// TIA Portal V19 export
FUNCTION "INPUT" : Void   // FC1, LAD
{ S7_Optimized_Access := 'TRUE' }
// stored: SetENOAutomatically false
BEGIN

REGION Network 1: "EMG STOP"
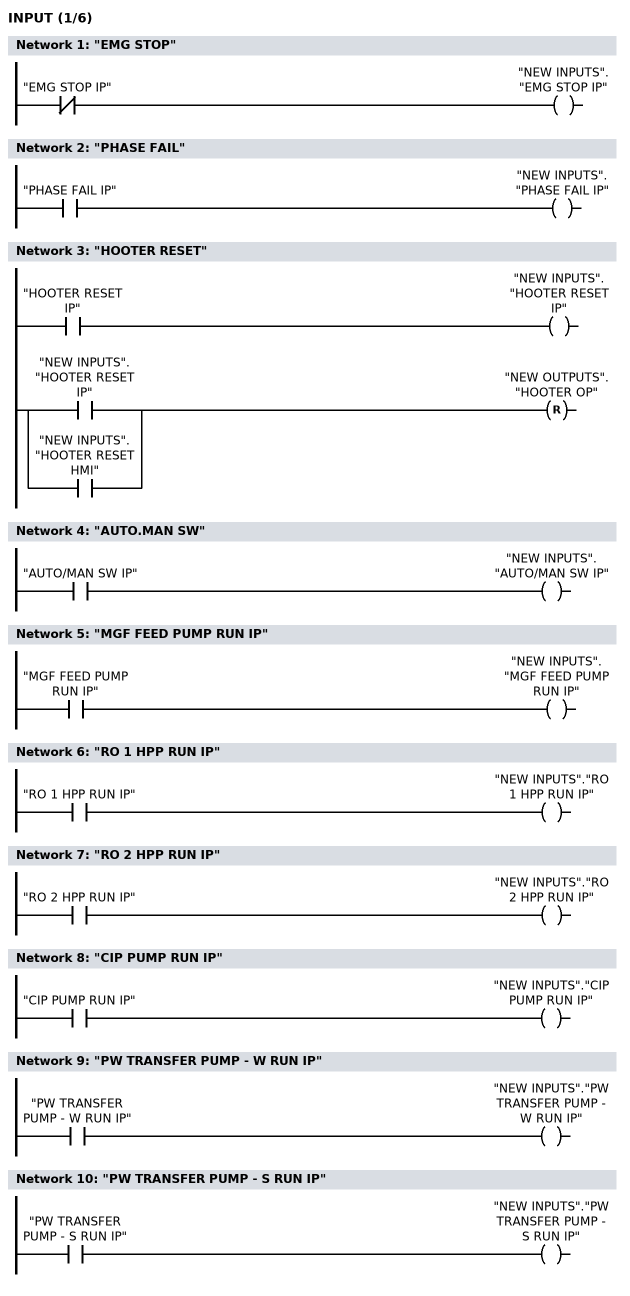
   RUNG wire#powerrail
      I_Contact( "EMG STOP IP" )
      Coil( "NEW INPUTS"."EMG STOP IP" )
   END_RUNG
   // the same network as SCL:
   "NEW INPUTS"."EMG STOP IP" := NOT "EMG STOP IP";
END_REGION

REGION Network 2: "PHASE FAIL"
   RUNG wire#powerrail
      Contact( "PHASE FAIL IP" )
      Coil( "NEW INPUTS"."PHASE FAIL IP" )
   END_RUNG
   // the same network as SCL:
   "NEW INPUTS"."PHASE FAIL IP" := "PHASE FAIL IP";
END_REGION

REGION Network 3: "HOOTER RESET"
   RUNG wire#powerrail
      Contact( "HOOTER RESET IP" )
      Coil( "NEW INPUTS"."HOOTER RESET IP" )
   END_RUNG
   RUNG wire#powerrail
      Contact( "NEW INPUTS"."HOOTER RESET IP" )
      wire#w1
      R_Coil( "NEW OUTPUTS"."HOOTER OP" )
   END_RUNG
   RUNG wire#powerrail
      Contact( "NEW INPUTS"."HOOTER RESET HMI" )
   END_RUNG wire#w1
   // the same network as SCL:
   "NEW INPUTS"."HOOTER RESET IP" := "HOOTER RESET IP";
   IF "NEW INPUTS"."HOOTER RESET IP" OR "NEW INPUTS"."HOOTER RESET HMI" THEN
       "NEW OUTPUTS"."HOOTER OP" := FALSE;
   END_IF;
END_REGION

REGION Network 4: "AUTO.MAN SW"
   RUNG wire#powerrail
      Contact( "AUTO/MAN SW IP" )
      Coil( "NEW INPUTS"."AUTO/MAN SW IP" )
   END_RUNG
   // the same network as SCL:
   "NEW INPUTS"."AUTO/MAN SW IP" := "AUTO/MAN SW IP";
END_REGION

REGION Network 5: "MGF FEED PUMP RUN IP"
   RUNG wire#powerrail
      Contact( "MGF FEED PUMP RUN IP" )
      Coil( "NEW INPUTS"."MGF FEED PUMP RUN IP" )
   END_RUNG
   // the same network as SCL:
   "NEW INPUTS"."MGF FEED PUMP RUN IP" := "MGF FEED PUMP RUN IP";
END_REGION

REGION Network 6: "RO 1 HPP RUN IP"
   RUNG wire#powerrail
      Contact( "RO 1 HPP RUN IP" )
      Coil( "NEW INPUTS"."RO 1 HPP RUN IP" )
   END_RUNG
   // the same network as SCL:
   "NEW INPUTS"."RO 1 HPP RUN IP" := "RO 1 HPP RUN IP";
END_REGION

REGION Network 7: "RO 2 HPP RUN IP"
   RUNG wire#powerrail
      Contact( "RO 2 HPP RUN IP" )
      Coil( "NEW INPUTS"."RO 2 HPP RUN IP" )
   END_RUNG
   // the same network as SCL:
   "NEW INPUTS"."RO 2 HPP RUN IP" := "RO 2 HPP RUN IP";
END_REGION

REGION Network 8: "CIP PUMP RUN IP"
   RUNG wire#powerrail
      Contact( "CIP PUMP RUN IP" )
      Coil( "NEW INPUTS"."CIP PUMP RUN IP" )
   END_RUNG
   // the same network as SCL:
   "NEW INPUTS"."CIP PUMP RUN IP" := "CIP PUMP RUN IP";
END_REGION

REGION Network 9: "PW TRANSFER PUMP - W RUN IP"
   RUNG wire#powerrail
      Contact( "PW TRANSFER PUMP - W RUN IP" )
      Coil( "NEW INPUTS"."PW TRANSFER PUMP - W RUN IP" )
   END_RUNG
   // the same network as SCL:
   "NEW INPUTS"."PW TRANSFER PUMP - W RUN IP" := "PW TRANSFER PUMP - W RUN IP";
END_REGION

REGION Network 10: "PW TRANSFER PUMP - S RUN IP"
   RUNG wire#powerrail
      Contact( "PW TRANSFER PUMP - S RUN IP" )
      Coil( "NEW INPUTS"."PW TRANSFER PUMP - S RUN IP" )
   END_RUNG
   // the same network as SCL:
   "NEW INPUTS"."PW TRANSFER PUMP - S RUN IP" := "PW TRANSFER PUMP - S RUN IP";
END_REGION

REGION Network 11: PW TRANSFER W/P
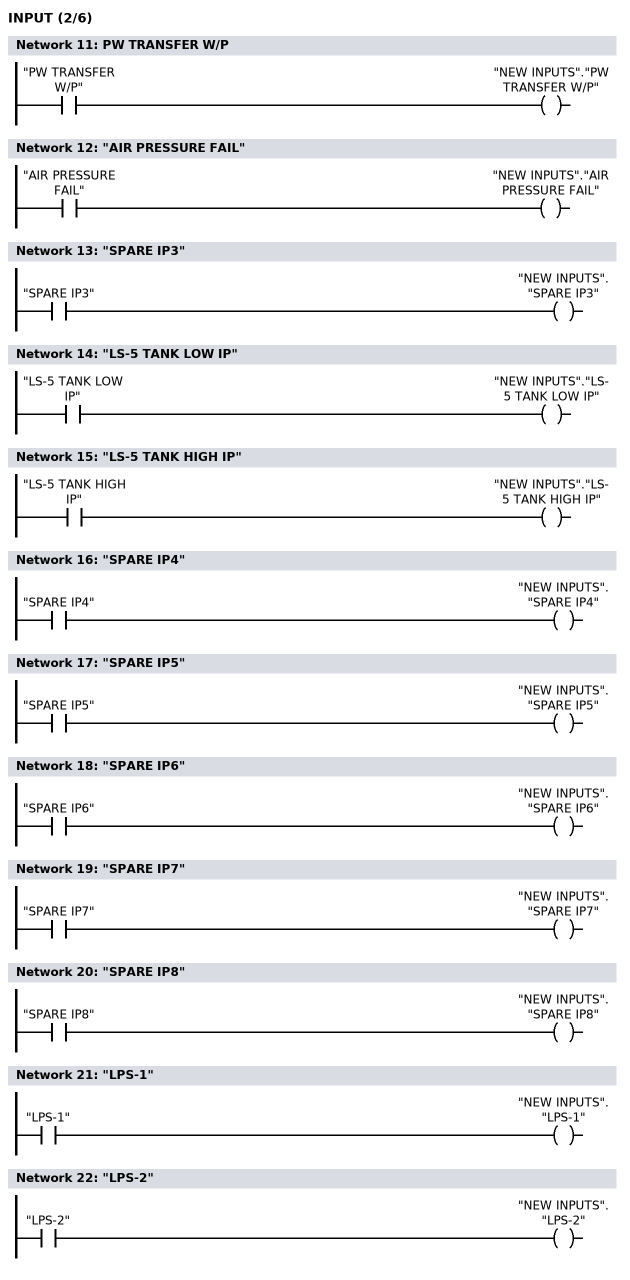
   RUNG wire#powerrail
      Contact( "PW TRANSFER W/P" )
      Coil( "NEW INPUTS"."PW TRANSFER W/P" )
   END_RUNG
   // the same network as SCL:
   "NEW INPUTS"."PW TRANSFER W/P" := "PW TRANSFER W/P";
END_REGION

REGION Network 12: "AIR PRESSURE FAIL"
   RUNG wire#powerrail
      Contact( "AIR PRESSURE FAIL" )
      Coil( "NEW INPUTS"."AIR PRESSURE FAIL" )
   END_RUNG
   // the same network as SCL:
   "NEW INPUTS"."AIR PRESSURE FAIL" := "AIR PRESSURE FAIL";
END_REGION

REGION Network 13: "SPARE IP3"
   RUNG wire#powerrail
      Contact( "SPARE IP3" )
      Coil( "NEW INPUTS"."SPARE IP3" )
   END_RUNG
   // the same network as SCL:
   "NEW INPUTS"."SPARE IP3" := "SPARE IP3";
END_REGION

REGION Network 14: "LS-5 TANK LOW IP"
   RUNG wire#powerrail
      Contact( "LS-5 TANK LOW IP" )
      Coil( "NEW INPUTS"."LS-5 TANK LOW IP" )
   END_RUNG
   // the same network as SCL:
   "NEW INPUTS"."LS-5 TANK LOW IP" := "LS-5 TANK LOW IP";
END_REGION

REGION Network 15: "LS-5 TANK HIGH IP"
   RUNG wire#powerrail
      Contact( "LS-5 TANK HIGH IP" )
      Coil( "NEW INPUTS"."LS-5 TANK HIGH IP" )
   END_RUNG
   // the same network as SCL:
   "NEW INPUTS"."LS-5 TANK HIGH IP" := "LS-5 TANK HIGH IP";
END_REGION

REGION Network 16: "SPARE IP4"
   RUNG wire#powerrail
      Contact( "SPARE IP4" )
      Coil( "NEW INPUTS"."SPARE IP4" )
   END_RUNG
   // the same network as SCL:
   "NEW INPUTS"."SPARE IP4" := "SPARE IP4";
END_REGION

REGION Network 17: "SPARE IP5"
   RUNG wire#powerrail
      Contact( "SPARE IP5" )
      Coil( "NEW INPUTS"."SPARE IP5" )
   END_RUNG
   // the same network as SCL:
   "NEW INPUTS"."SPARE IP5" := "SPARE IP5";
END_REGION

REGION Network 18: "SPARE IP6"
   RUNG wire#powerrail
      Contact( "SPARE IP6" )
      Coil( "NEW INPUTS"."SPARE IP6" )
   END_RUNG
   // the same network as SCL:
   "NEW INPUTS"."SPARE IP6" := "SPARE IP6";
END_REGION

REGION Network 19: "SPARE IP7"
   RUNG wire#powerrail
      Contact( "SPARE IP7" )
      Coil( "NEW INPUTS"."SPARE IP7" )
   END_RUNG
   // the same network as SCL:
   "NEW INPUTS"."SPARE IP7" := "SPARE IP7";
END_REGION

REGION Network 20: "SPARE IP8"
   RUNG wire#powerrail
      Contact( "SPARE IP8" )
      Coil( "NEW INPUTS"."SPARE IP8" )
   END_RUNG
   // the same network as SCL:
   "NEW INPUTS"."SPARE IP8" := "SPARE IP8";
END_REGION

REGION Network 21: "LPS-1"
   RUNG wire#powerrail
      Contact( "LPS-1" )
      Coil( "NEW INPUTS"."LPS-1" )
   END_RUNG
   // the same network as SCL:
   "NEW INPUTS"."LPS-1" := "LPS-1";
END_REGION

REGION Network 22: "LPS-2"
   RUNG wire#powerrail
      Contact( "LPS-2" )
      Coil( "NEW INPUTS"."LPS-2" )
   END_RUNG
   // the same network as SCL:
   "NEW INPUTS"."LPS-2" := "LPS-2";
END_REGION

REGION Network 23: "MGF V-1 OPEN FB"
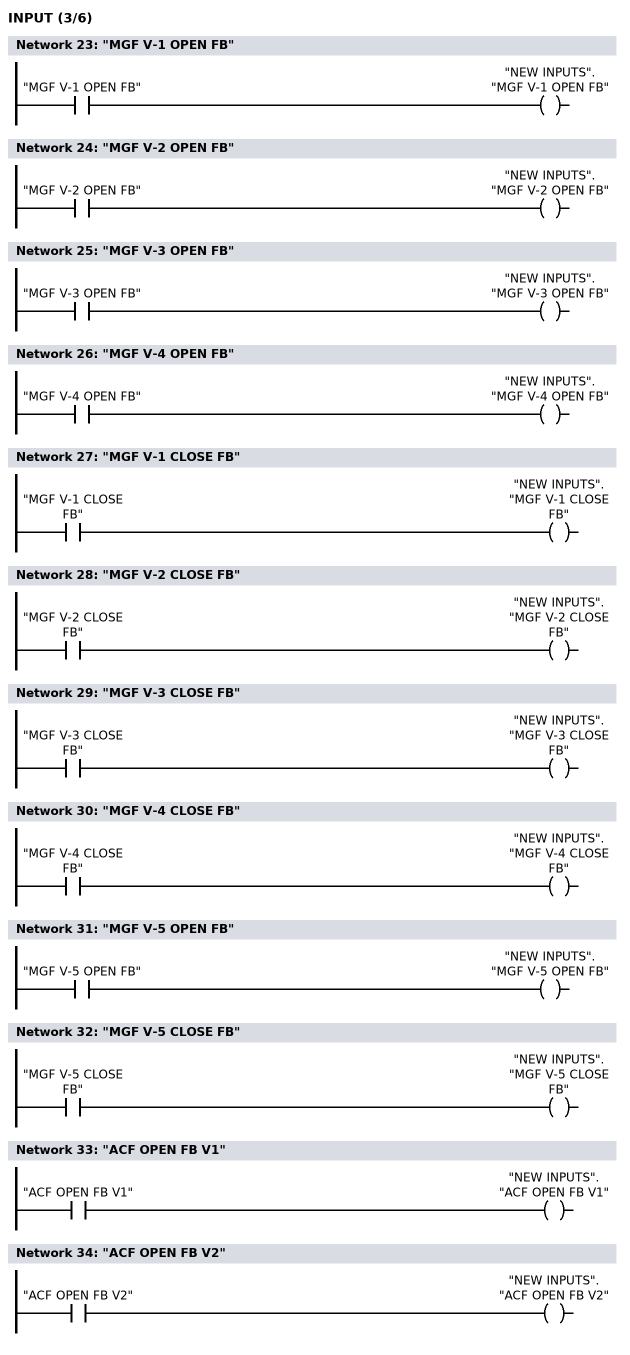
   RUNG wire#powerrail
      Contact( "MGF V-1 OPEN FB" )
      Coil( "NEW INPUTS"."MGF V-1 OPEN FB" )
   END_RUNG
   // the same network as SCL:
   "NEW INPUTS"."MGF V-1 OPEN FB" := "MGF V-1 OPEN FB";
END_REGION

REGION Network 24: "MGF V-2 OPEN FB"
   RUNG wire#powerrail
      Contact( "MGF V-2 OPEN FB" )
      Coil( "NEW INPUTS"."MGF V-2 OPEN FB" )
   END_RUNG
   // the same network as SCL:
   "NEW INPUTS"."MGF V-2 OPEN FB" := "MGF V-2 OPEN FB";
END_REGION

REGION Network 25: "MGF V-3 OPEN FB"
   RUNG wire#powerrail
      Contact( "MGF V-3 OPEN FB" )
      Coil( "NEW INPUTS"."MGF V-3 OPEN FB" )
   END_RUNG
   // the same network as SCL:
   "NEW INPUTS"."MGF V-3 OPEN FB" := "MGF V-3 OPEN FB";
END_REGION

REGION Network 26: "MGF V-4 OPEN FB"
   RUNG wire#powerrail
      Contact( "MGF V-4 OPEN FB" )
      Coil( "NEW INPUTS"."MGF V-4 OPEN FB" )
   END_RUNG
   // the same network as SCL:
   "NEW INPUTS"."MGF V-4 OPEN FB" := "MGF V-4 OPEN FB";
END_REGION

REGION Network 27: "MGF V-1 CLOSE FB"
   RUNG wire#powerrail
      Contact( "MGF V-1 CLOSE FB" )
      Coil( "NEW INPUTS"."MGF V-1 CLOSE FB" )
   END_RUNG
   // the same network as SCL:
   "NEW INPUTS"."MGF V-1 CLOSE FB" := "MGF V-1 CLOSE FB";
END_REGION

REGION Network 28: "MGF V-2 CLOSE FB"
   RUNG wire#powerrail
      Contact( "MGF V-2 CLOSE FB" )
      Coil( "NEW INPUTS"."MGF V-2 CLOSE FB" )
   END_RUNG
   // the same network as SCL:
   "NEW INPUTS"."MGF V-2 CLOSE FB" := "MGF V-2 CLOSE FB";
END_REGION

REGION Network 29: "MGF V-3 CLOSE FB"
   RUNG wire#powerrail
      Contact( "MGF V-3 CLOSE FB" )
      Coil( "NEW INPUTS"."MGF V-3 CLOSE FB" )
   END_RUNG
   // the same network as SCL:
   "NEW INPUTS"."MGF V-3 CLOSE FB" := "MGF V-3 CLOSE FB";
END_REGION

REGION Network 30: "MGF V-4 CLOSE FB"
   RUNG wire#powerrail
      Contact( "MGF V-4 CLOSE FB" )
      Coil( "NEW INPUTS"."MGF V-4 CLOSE FB" )
   END_RUNG
   // the same network as SCL:
   "NEW INPUTS"."MGF V-4 CLOSE FB" := "MGF V-4 CLOSE FB";
END_REGION

REGION Network 31: "MGF V-5 OPEN FB"
   RUNG wire#powerrail
      Contact( "MGF V-5 OPEN FB" )
      Coil( "NEW INPUTS"."MGF V-5 OPEN FB" )
   END_RUNG
   // the same network as SCL:
   "NEW INPUTS"."MGF V-5 OPEN FB" := "MGF V-5 OPEN FB";
END_REGION

REGION Network 32: "MGF V-5 CLOSE FB"
   RUNG wire#powerrail
      Contact( "MGF V-5 CLOSE FB" )
      Coil( "NEW INPUTS"."MGF V-5 CLOSE FB" )
   END_RUNG
   // the same network as SCL:
   "NEW INPUTS"."MGF V-5 CLOSE FB" := "MGF V-5 CLOSE FB";
END_REGION

REGION Network 33: "ACF OPEN FB V1"
   RUNG wire#powerrail
      Contact( "ACF OPEN FB V1" )
      Coil( "NEW INPUTS"."ACF OPEN FB V1" )
   END_RUNG
   // the same network as SCL:
   "NEW INPUTS"."ACF OPEN FB V1" := "ACF OPEN FB V1";
END_REGION

REGION Network 34: "ACF OPEN FB V2"
   RUNG wire#powerrail
      Contact( "ACF OPEN FB V2" )
      Coil( "NEW INPUTS"."ACF OPEN FB V2" )
   END_RUNG
   // the same network as SCL:
   "NEW INPUTS"."ACF OPEN FB V2" := "ACF OPEN FB V2";
END_REGION

REGION Network 35: "ACF OPEN FB V3"
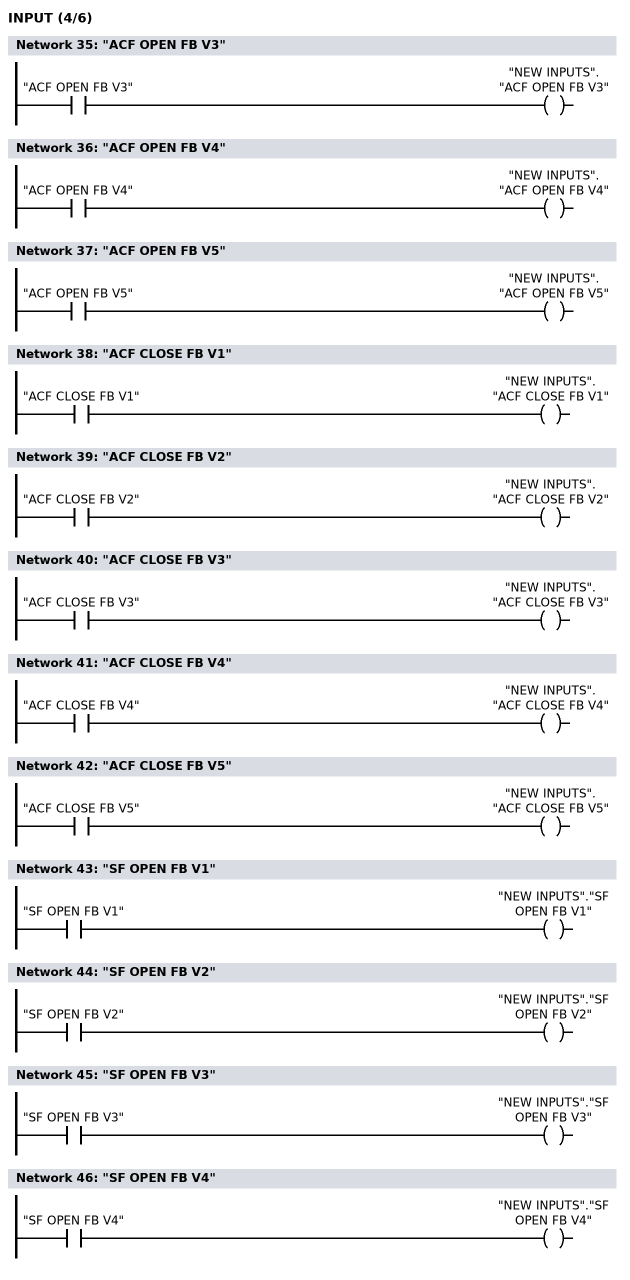
   RUNG wire#powerrail
      Contact( "ACF OPEN FB V3" )
      Coil( "NEW INPUTS"."ACF OPEN FB V3" )
   END_RUNG
   // the same network as SCL:
   "NEW INPUTS"."ACF OPEN FB V3" := "ACF OPEN FB V3";
END_REGION

REGION Network 36: "ACF OPEN FB V4"
   RUNG wire#powerrail
      Contact( "ACF OPEN FB V4" )
      Coil( "NEW INPUTS"."ACF OPEN FB V4" )
   END_RUNG
   // the same network as SCL:
   "NEW INPUTS"."ACF OPEN FB V4" := "ACF OPEN FB V4";
END_REGION

REGION Network 37: "ACF OPEN FB V5"
   RUNG wire#powerrail
      Contact( "ACF OPEN FB V5" )
      Coil( "NEW INPUTS"."ACF OPEN FB V5" )
   END_RUNG
   // the same network as SCL:
   "NEW INPUTS"."ACF OPEN FB V5" := "ACF OPEN FB V5";
END_REGION

REGION Network 38: "ACF CLOSE FB V1"
   RUNG wire#powerrail
      Contact( "ACF CLOSE FB V1" )
      Coil( "NEW INPUTS"."ACF CLOSE FB V1" )
   END_RUNG
   // the same network as SCL:
   "NEW INPUTS"."ACF CLOSE FB V1" := "ACF CLOSE FB V1";
END_REGION

REGION Network 39: "ACF CLOSE FB V2"
   RUNG wire#powerrail
      Contact( "ACF CLOSE FB V2" )
      Coil( "NEW INPUTS"."ACF CLOSE FB V2" )
   END_RUNG
   // the same network as SCL:
   "NEW INPUTS"."ACF CLOSE FB V2" := "ACF CLOSE FB V2";
END_REGION

REGION Network 40: "ACF CLOSE FB V3"
   RUNG wire#powerrail
      Contact( "ACF CLOSE FB V3" )
      Coil( "NEW INPUTS"."ACF CLOSE FB V3" )
   END_RUNG
   // the same network as SCL:
   "NEW INPUTS"."ACF CLOSE FB V3" := "ACF CLOSE FB V3";
END_REGION

REGION Network 41: "ACF CLOSE FB V4"
   RUNG wire#powerrail
      Contact( "ACF CLOSE FB V4" )
      Coil( "NEW INPUTS"."ACF CLOSE FB V4" )
   END_RUNG
   // the same network as SCL:
   "NEW INPUTS"."ACF CLOSE FB V4" := "ACF CLOSE FB V4";
END_REGION

REGION Network 42: "ACF CLOSE FB V5"
   RUNG wire#powerrail
      Contact( "ACF CLOSE FB V5" )
      Coil( "NEW INPUTS"."ACF CLOSE FB V5" )
   END_RUNG
   // the same network as SCL:
   "NEW INPUTS"."ACF CLOSE FB V5" := "ACF CLOSE FB V5";
END_REGION

REGION Network 43: "SF OPEN FB V1"
   RUNG wire#powerrail
      Contact( "SF OPEN FB V1" )
      Coil( "NEW INPUTS"."SF OPEN FB V1" )
   END_RUNG
   // the same network as SCL:
   "NEW INPUTS"."SF OPEN FB V1" := "SF OPEN FB V1";
END_REGION

REGION Network 44: "SF OPEN FB V2"
   RUNG wire#powerrail
      Contact( "SF OPEN FB V2" )
      Coil( "NEW INPUTS"."SF OPEN FB V2" )
   END_RUNG
   // the same network as SCL:
   "NEW INPUTS"."SF OPEN FB V2" := "SF OPEN FB V2";
END_REGION

REGION Network 45: "SF OPEN FB V3"
   RUNG wire#powerrail
      Contact( "SF OPEN FB V3" )
      Coil( "NEW INPUTS"."SF OPEN FB V3" )
   END_RUNG
   // the same network as SCL:
   "NEW INPUTS"."SF OPEN FB V3" := "SF OPEN FB V3";
END_REGION

REGION Network 46: "SF OPEN FB V4"
   RUNG wire#powerrail
      Contact( "SF OPEN FB V4" )
      Coil( "NEW INPUTS"."SF OPEN FB V4" )
   END_RUNG
   // the same network as SCL:
   "NEW INPUTS"."SF OPEN FB V4" := "SF OPEN FB V4";
END_REGION

REGION Network 47: "SF OPEN FB V5"
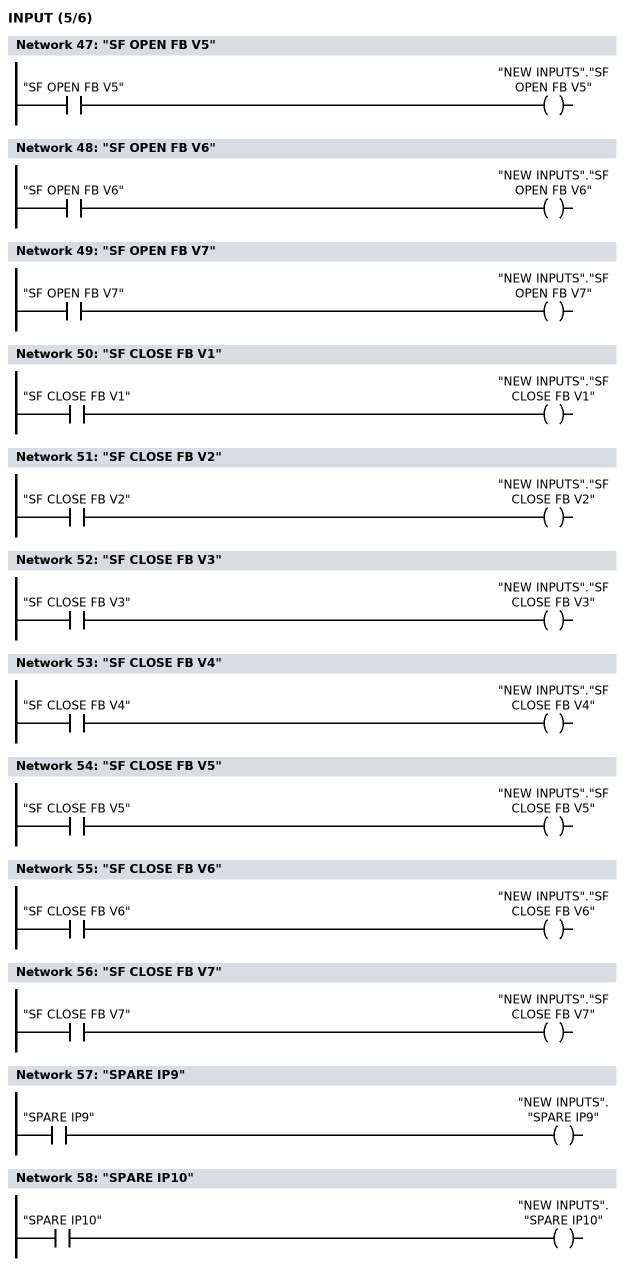
   RUNG wire#powerrail
      Contact( "SF OPEN FB V5" )
      Coil( "NEW INPUTS"."SF OPEN FB V5" )
   END_RUNG
   // the same network as SCL:
   "NEW INPUTS"."SF OPEN FB V5" := "SF OPEN FB V5";
END_REGION

REGION Network 48: "SF OPEN FB V6"
   RUNG wire#powerrail
      Contact( "SF OPEN FB V6" )
      Coil( "NEW INPUTS"."SF OPEN FB V6" )
   END_RUNG
   // the same network as SCL:
   "NEW INPUTS"."SF OPEN FB V6" := "SF OPEN FB V6";
END_REGION

REGION Network 49: "SF OPEN FB V7"
   RUNG wire#powerrail
      Contact( "SF OPEN FB V7" )
      Coil( "NEW INPUTS"."SF OPEN FB V7" )
   END_RUNG
   // the same network as SCL:
   "NEW INPUTS"."SF OPEN FB V7" := "SF OPEN FB V7";
END_REGION

REGION Network 50: "SF CLOSE FB V1"
   RUNG wire#powerrail
      Contact( "SF CLOSE FB V1" )
      Coil( "NEW INPUTS"."SF CLOSE FB V1" )
   END_RUNG
   // the same network as SCL:
   "NEW INPUTS"."SF CLOSE FB V1" := "SF CLOSE FB V1";
END_REGION

REGION Network 51: "SF CLOSE FB V2"
   RUNG wire#powerrail
      Contact( "SF CLOSE FB V2" )
      Coil( "NEW INPUTS"."SF CLOSE FB V2" )
   END_RUNG
   // the same network as SCL:
   "NEW INPUTS"."SF CLOSE FB V2" := "SF CLOSE FB V2";
END_REGION

REGION Network 52: "SF CLOSE FB V3"
   RUNG wire#powerrail
      Contact( "SF CLOSE FB V3" )
      Coil( "NEW INPUTS"."SF CLOSE FB V3" )
   END_RUNG
   // the same network as SCL:
   "NEW INPUTS"."SF CLOSE FB V3" := "SF CLOSE FB V3";
END_REGION

REGION Network 53: "SF CLOSE FB V4"
   RUNG wire#powerrail
      Contact( "SF CLOSE FB V4" )
      Coil( "NEW INPUTS"."SF CLOSE FB V4" )
   END_RUNG
   // the same network as SCL:
   "NEW INPUTS"."SF CLOSE FB V4" := "SF CLOSE FB V4";
END_REGION

REGION Network 54: "SF CLOSE FB V5"
   RUNG wire#powerrail
      Contact( "SF CLOSE FB V5" )
      Coil( "NEW INPUTS"."SF CLOSE FB V5" )
   END_RUNG
   // the same network as SCL:
   "NEW INPUTS"."SF CLOSE FB V5" := "SF CLOSE FB V5";
END_REGION

REGION Network 55: "SF CLOSE FB V6"
   RUNG wire#powerrail
      Contact( "SF CLOSE FB V6" )
      Coil( "NEW INPUTS"."SF CLOSE FB V6" )
   END_RUNG
   // the same network as SCL:
   "NEW INPUTS"."SF CLOSE FB V6" := "SF CLOSE FB V6";
END_REGION

REGION Network 56: "SF CLOSE FB V7"
   RUNG wire#powerrail
      Contact( "SF CLOSE FB V7" )
      Coil( "NEW INPUTS"."SF CLOSE FB V7" )
   END_RUNG
   // the same network as SCL:
   "NEW INPUTS"."SF CLOSE FB V7" := "SF CLOSE FB V7";
END_REGION

REGION Network 57: "SPARE IP9"
   RUNG wire#powerrail
      Contact( "SPARE IP9" )
      Coil( "NEW INPUTS"."SPARE IP9" )
   END_RUNG
   // the same network as SCL:
   "NEW INPUTS"."SPARE IP9" := "SPARE IP9";
END_REGION

REGION Network 58: "SPARE IP10"
   RUNG wire#powerrail
      Contact( "SPARE IP10" )
      Coil( "NEW INPUTS"."SPARE IP10" )
   END_RUNG
   // the same network as SCL:
   "NEW INPUTS"."SPARE IP10" := "SPARE IP10";
END_REGION

REGION Network 59: "SPARE IP11"
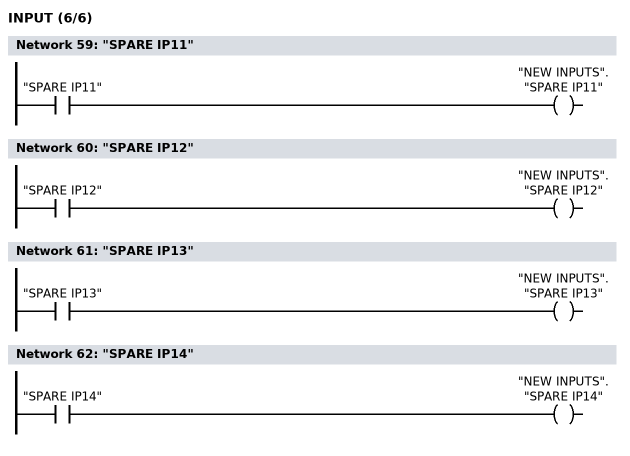
   RUNG wire#powerrail
      Contact( "SPARE IP11" )
      Coil( "NEW INPUTS"."SPARE IP11" )
   END_RUNG
   // the same network as SCL:
   "NEW INPUTS"."SPARE IP11" := "SPARE IP11";
END_REGION

REGION Network 60: "SPARE IP12"
   RUNG wire#powerrail
      Contact( "SPARE IP12" )
      Coil( "NEW INPUTS"."SPARE IP12" )
   END_RUNG
   // the same network as SCL:
   "NEW INPUTS"."SPARE IP12" := "SPARE IP12";
END_REGION

REGION Network 61: "SPARE IP13"
   RUNG wire#powerrail
      Contact( "SPARE IP13" )
      Coil( "NEW INPUTS"."SPARE IP13" )
   END_RUNG
   // the same network as SCL:
   "NEW INPUTS"."SPARE IP13" := "SPARE IP13";
END_REGION

REGION Network 62: "SPARE IP14"
   RUNG wire#powerrail
      Contact( "SPARE IP14" )
      Coil( "NEW INPUTS"."SPARE IP14" )
   END_RUNG
   // the same network as SCL:
   "NEW INPUTS"."SPARE IP14" := "SPARE IP14";
END_REGION
END_FUNCTION
